{attribute 'GeneratedUsingTerminal: EL6201-0000-0017'}
{attribute addProperty BoxType "EL6201-0000-0017"}
{attribute addProperty Id "Slave_31A_DI0BOOL1Slave_31A_DI1BOOL1Slave_31A_DI2BOOL1Slave_31A_DI3BOOL1Slave_31B_DI0BOOL1Slave_31B_DI1BOOL1Slave_31B_DI2BOOL1Slave_31B_DI3BOOL1"}
{attribute addProperty CRC "3389966400"}
{attribute addProperty Size "8"}
TYPE Slave_31_Inputs_CA0EC840 :
STRUCT
	{attribute addProperty Name "Slave_31A_DI0"}
	Slave_31A_DI0 : BOOL;
	{attribute addProperty Name "Slave_31A_DI1"}
	Slave_31A_DI1 : BOOL;
	{attribute addProperty Name "Slave_31A_DI2"}
	Slave_31A_DI2 : BOOL;
	{attribute addProperty Name "Slave_31A_DI3"}
	Slave_31A_DI3 : BOOL;
	{attribute addProperty Name "Slave_31B_DI0"}
	Slave_31B_DI0 : BOOL;
	{attribute addProperty Name "Slave_31B_DI1"}
	Slave_31B_DI1 : BOOL;
	{attribute addProperty Name "Slave_31B_DI2"}
	Slave_31B_DI2 : BOOL;
	{attribute addProperty Name "Slave_31B_DI3"}
	Slave_31B_DI3 : BOOL;
END_STRUCT
END_TYPE

(* stored: Version 1.2.0.0, ProductVersion 3.1.4024.9
   DUT Slave_31_Inputs_CA0EC840: Id {e51d79e0-b16f-4aed-970d-6eab61dd4ab0} *)
